INTERFACE I_LoggerConfig

// Gets the logger configuration - should not be edited, use .Configure() method to apply configuration.
{attribute 'monitoring':='call'}
PROPERTY Configuration : REFERENCE TO ST_LoggerConfiguration
GET
END_GET
END_PROPERTY

METHOD Configure : I_LoggerConfigBuilder
END_METHOD

END_INTERFACE

(* stored: Version 1.1.0.1, ProductVersion 3.1.4024.15
   Itf I_LoggerConfig: Id {2ba2c81e-fc2d-0294-2104-7f3b7e99342f}
   Property Configuration: Id {edcd145b-ef6d-0d72-1fa0-8765e3596706}
   Get Get: Id {45e35ee2-16ef-0bcc-29de-9617a79dbbb8}
   Method Configure: Id {11ca3005-1876-025b-2a7c-452747fb79b2} *)
